INTERFACE I_FloatArg EXTENDS I_Arg

PROPERTY Val : LREAL
GET
END_GET
END_PROPERTY

END_INTERFACE

(* stored: Version 1.1.0.1
   Itf I_FloatArg: Id {7a9d8070-f2e7-4e82-9412-c14723403e71}
   Property Val: Id {75a1495a-cd7c-4507-a8a7-53186b9fe88f}
   Get Get: Id {297213ed-995a-47b6-80ea-9224306c344b} *)
